// TIA Portal V20 export
DATA_BLOCK "Config"   // DB83
// stored: Access Published, MemoryReserve 100, Namespace Unit1.Em8
   VAR
      em : "LAF_typeEmConfiguration";   // Configuration of EM Parameters
      axis : Array[0.._.U1EM8_JOB03] of DB_ANY;
      cmHipotThicknessSafetyPin : "LBC_typeDigitalSignalConfiguration";
      cmHipotThicknessJRDetect : "LBC_typeDigitalSignalConfiguration";
   END_VAR
   VAR RETAIN
      cmThicknessAxisZ : "LBC_typeAxis64PosConfiguration";
   END_VAR
   VAR
      cmHipotThicknessStageLiftFrontUpDown : "LBC_typeTwoWayActuatorConfiguration";
      cmHipotThicknessStageLiftRearUpDown : "LBC_typeTwoWayActuatorConfiguration";
      cmHipotTabContactorBwdFwd : "LBC_typeTwoWayActuatorConfiguration";
      cmHipotTabContactorLeftOpenClose : "LBC_typeTwoWayActuatorConfiguration";
      cmHipotTabContactorRightOpenClose : "LBC_typeTwoWayActuatorConfiguration";
      cmHipotThicknessStageLiftAllUpDown : "LBC_typeTwoWayActuatorConfiguration";
      cmHipotThicknessServoPress : "LER_typeServoPressConfiguration";
      cmThicknessControl : "LER_typeThicknessConfiguration";
      cmHipotControl : "LER_typeHipotConfiguration";
      softcam : Struct
         ThicknessAxisZ : "LER_typeSoftCamInterface";
      END_STRUCT;
   END_VAR
BEGIN
   em.referenceDesignator.parent := WSTRING#'U1';
   em.referenceDesignator.relative := WSTRING#'EM0';
   cmThicknessAxisZ.referenceDesignator := WSTRING#'HI-POT & THICKNESS Z-Axis';
   cmHipotThicknessStageLiftFrontUpDown.referenceDesignator := WSTRING#'STAGE LIFT FRONT';
   cmHipotThicknessStageLiftFrontUpDown.monitoringDiscrepancy := T#5s;
   cmHipotThicknessStageLiftRearUpDown.referenceDesignator := WSTRING#'STAGE LIFT REAR';
   cmHipotThicknessStageLiftRearUpDown.monitoringDiscrepancy := T#5s;
   cmHipotTabContactorBwdFwd.referenceDesignator := WSTRING#'TAB CONTACTOR';
   cmHipotTabContactorBwdFwd.monitoringDiscrepancy := T#5s;
   cmHipotTabContactorLeftOpenClose.referenceDesignator := WSTRING#'TAB CONTACTOR LEFT';
   cmHipotTabContactorLeftOpenClose.monitoringDiscrepancy := T#5s;
   cmHipotTabContactorRightOpenClose.referenceDesignator := WSTRING#'TAB CONTACTOR RIGHT';
   cmHipotTabContactorRightOpenClose.monitoringDiscrepancy := T#5s;
   cmHipotThicknessStageLiftAllUpDown.referenceDesignator := WSTRING#'Stage';
   cmHipotThicknessStageLiftAllUpDown.monitoringDiscrepancy := T#5s;
   cmHipotThicknessServoPress.hwID."220ByteIn" := 661;
   cmHipotThicknessServoPress.hwID."220ByteOut" := 660;
   cmThicknessControl.hwID.interfaceControllerID := 420;
   cmThicknessControl.hwID.ampID[0] := 421;
   cmThicknessControl.hwID.ampID[1] := 422;
   cmThicknessControl.hwID.ampID[2] := 423;
   cmThicknessControl.hwID.ampID[3] := 424;
   cmHipotControl.port := 1054;
END_DATA_BLOCK
